// Mitsubishi GX Works2 project: plc_group_22   PLC: FX3G

// global labels: Global1
VAR_GLOBAL
  startDayButton AT X010 : BOOL;
  workingDay AT Y010 : BOOL;
  emergencyButon AT X007 : BOOL;
  startSwich AT X010 : BOOL;
  startSwitch AT X010 : BOOL;
  initialClementine AT D1102 : REAL;
END_VAR
VAR_GLOBAL CONSTANT
  one : REAL := 1;
END_VAR
VAR_GLOBAL
  initialPomelo AT D1104 : REAL;
END_VAR
VAR_GLOBAL CONSTANT
  two : REAL := 2;
END_VAR
VAR_GLOBAL
  initialOrange AT D1100 : REAL;
  enoughOranges AT M0 : BOOL;
  enoughClementine AT M1 : BOOL;
  enoughPomelo AT M2 : BOOL;
  noOranges AT M3 : BOOL;
  noClementine AT M4 : BOOL;
  noPomelos AT M5 : BOOL;
  blink AT M6 : BOOL;
  FIC AT M7 : BOOL;
END_VAR
VAR_GLOBAL CONSTANT
  time30 : INT := 30;
END_VAR
VAR_GLOBAL
  tc1 AT TC1 : BOOL;
END_VAR
VAR_GLOBAL CONSTANT
  time3 : INT := 3;
END_VAR
VAR_GLOBAL
  tc2 AT TC2 : BOOL;
  tc3 AT TC3 : BOOL;
  ts1 AT TS1 : BOOL;
  finale AT M11 : BOOL;
  ts3 AT TS3 : BOOL;
  FIc1 AT M20 : BOOL;
  temp AT M22 : BOOL;
  hold1 AT M23 : BOOL;
  startWash AT X002 : BOOL;
  tc4 AT TC4 : BOOL;
  ts4 AT TS4 : BOOL;
  washing AT Y005 : BOOL;
  storageOrange AT D1106 : REAL;
  storageClementine AT D1108 : REAL;
  storagePomelo AT D1110 : REAL;
  batchSize AT D1112 : REAL;
END_VAR
VAR_GLOBAL CONSTANT
  FIfthy : REAL := 50;
  zero : REAL;
END_VAR
VAR_GLOBAL
  orangeWashing AT D1114 : REAL;
  clementineWashing AT D1116 : REAL;
  pomeloWashing AT D1118 : REAL;
END_VAR
VAR_GLOBAL CONSTANT
  hundred : REAL := 100;
END_VAR
VAR_GLOBAL
  startCollection AT X001 : BOOL;
  collecting AT Y001 : BOOL;
  fruitContainer AT D1120 : REAL;
  juiceInProgress AT M12 : BOOL;
  startJuice AT X011 : BOOL;
  x11down AT M13 : BOOL;
  stopBlink AT TS2 : BOOL;
  blink1 AT M31 : BOOL;
  blink2 AT M32 : BOOL;
  startblink AT M33 : BOOL;
  closeDay AT M36 : BOOL;
  juiceLed1 AT Y002 : BOOL;
  juiceLed2 AT Y003 : BOOL;
  juiceContainer AT D1122 : REAL;
  endJuicing AT M40 : BOOL;
  counter0 AT CC0 : BOOL;
END_VAR
VAR_GLOBAL CONSTANT
  tow : INT := 2;
END_VAR
VAR_GLOBAL
  cs0 AT CS0 : BOOL;
END_VAR

// task Task_01 (event TRUE, interval 0, priority 31): POU_01

PROGRAM POU_01
(* structured ladder/FBD written out as ST: instructions are called as NAME(EN, inputs, outputs); _pN, _eN, _tN stand for wires *)
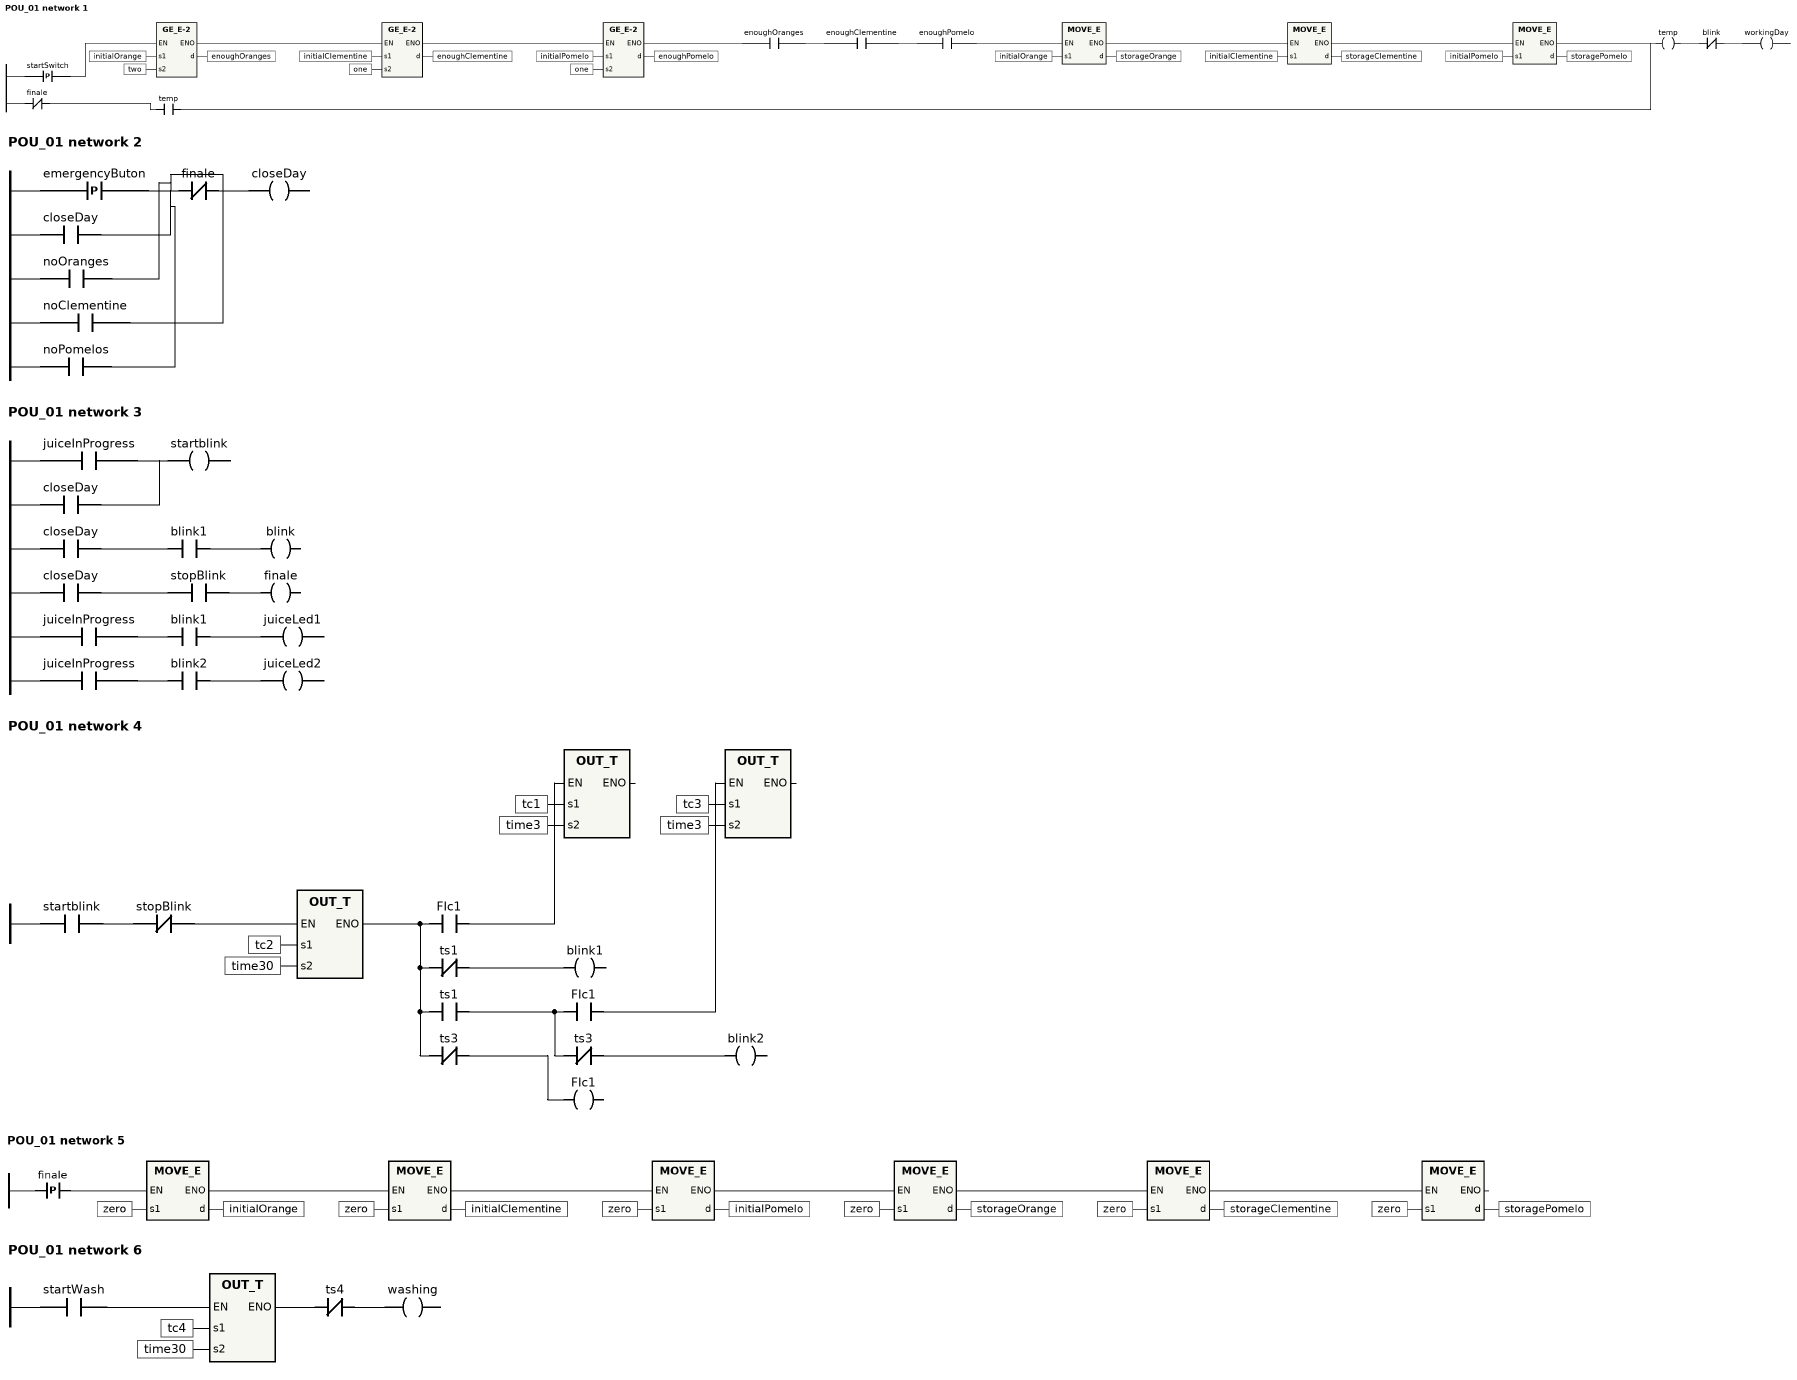
(* network 1 *)
_e1 := GE_E(LDP(TRUE, startSwitch), initialOrange, two, enoughOranges);
_e2 := GE_E(_e1, initialClementine, one, enoughClementine);
_e3 := GE_E(_e2, initialPomelo, one, enoughPomelo);
_e4 := MOVE_E(_e3 AND enoughOranges AND enoughClementine AND enoughPomelo, initialOrange, storageOrange);
_e5 := MOVE_E(_e4, initialClementine, storageClementine);
_e6 := MOVE_E(_e5, initialPomelo, storagePomelo);
_p7 := _e6 OR (NOT finale AND temp);
temp := _p7;
workingDay := _p7 AND NOT blink;
(* network 2 *)
closeDay := (LDP(TRUE, emergencyButon) OR closeDay OR noOranges OR noClementine OR noPomelos) AND NOT finale;
(* network 3 *)
startblink := juiceInProgress OR closeDay;
blink := closeDay AND blink1;
finale := closeDay AND stopBlink;
juiceLed1 := juiceInProgress AND blink1;
juiceLed2 := juiceInProgress AND blink2;
(* network 4 *)
_e1 := OUT_T(startblink AND NOT stopBlink, tc2, time30);
OUT_T(_e1 AND FIc1, tc1, time3);
blink1 := _e1 AND NOT ts1;
_p2 := _e1 AND ts1;
OUT_T(_p2 AND FIc1, tc3, time3);
blink2 := _p2 AND NOT ts3;
FIc1 := _e1 AND NOT ts3;
(* network 5 *)
_e1 := MOVE_E(LDP(TRUE, finale), zero, initialOrange);
_e2 := MOVE_E(_e1, zero, initialClementine);
_e3 := MOVE_E(_e2, zero, initialPomelo);
_e4 := MOVE_E(_e3, zero, storageOrange);
_e5 := MOVE_E(_e4, zero, storageClementine);
MOVE_E(_e5, zero, storagePomelo);
(* network 6 *)
_e1 := OUT_T(startWash, tc4, time30);
washing := _e1 AND NOT ts4;
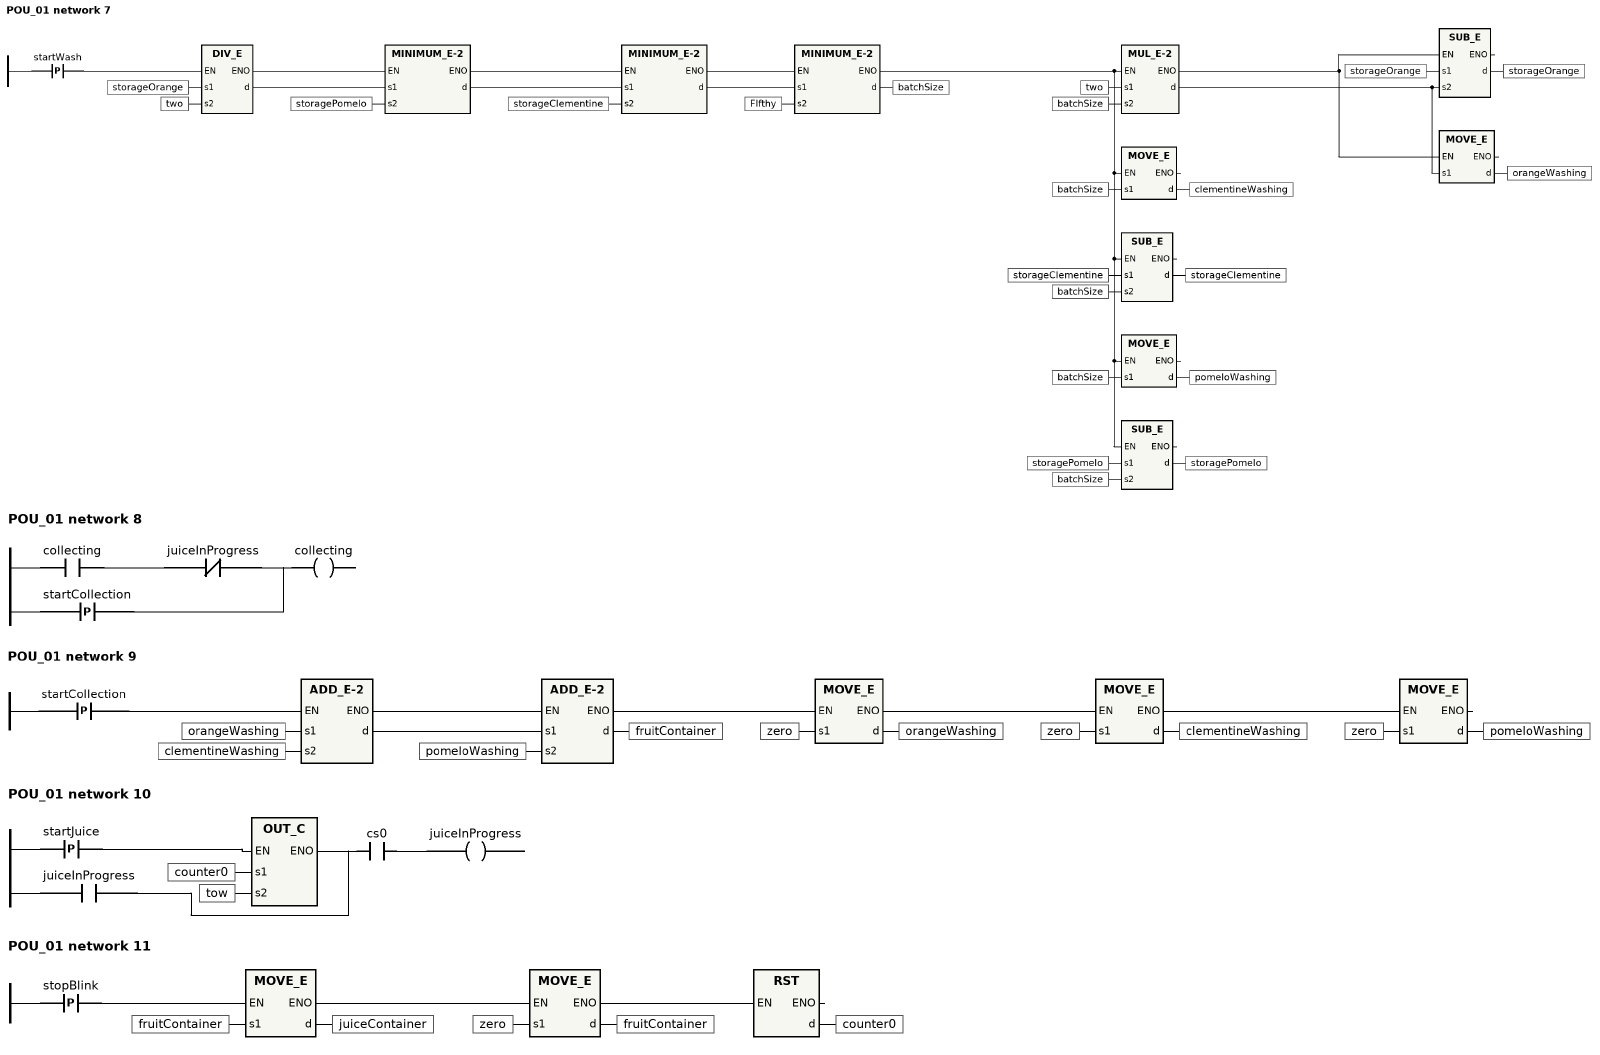
(* network 7 *)
_e2 := DIV_E(LDP(TRUE, startWash), storageOrange, two, _t1);
_e4 := MINIMUM_E(_e2, _t1, storagePomelo, _t3);
_e6 := MINIMUM_E(_e4, _t3, storageClementine, _t5);
_e7 := MINIMUM_E(_e6, _t5, FIfthy, batchSize);
_e9 := MUL_E(_e7, two, batchSize, _t8);
SUB_E(_e9, storageOrange, _t8, storageOrange);
MOVE_E(_e9, _t8, orangeWashing);
MOVE_E(_e7, batchSize, clementineWashing);
SUB_E(_e7, storageClementine, batchSize, storageClementine);
MOVE_E(_e7, batchSize, pomeloWashing);
SUB_E(_e7, storagePomelo, batchSize, storagePomelo);
(* network 8 *)
collecting := (collecting AND NOT juiceInProgress) OR LDP(TRUE, startCollection);
(* network 9 *)
_e2 := ADD_E(LDP(TRUE, startCollection), orangeWashing, clementineWashing, _t1);
_e3 := ADD_E(_e2, _t1, pomeloWashing, fruitContainer);
_e4 := MOVE_E(_e3, zero, orangeWashing);
_e5 := MOVE_E(_e4, zero, clementineWashing);
MOVE_E(_e5, zero, pomeloWashing);
(* network 10 *)
_e1 := OUT_C(LDP(TRUE, startJuice), counter0, tow);
juiceInProgress := (_e1 OR juiceInProgress) AND cs0;
(* network 11 *)
_e1 := MOVE_E(LDP(TRUE, stopBlink), fruitContainer, juiceContainer);
_e2 := MOVE_E(_e1, zero, fruitContainer);
RST(_e2, counter0);
END_PROGRAM
